FUNCTION_BLOCK ABSTRACT BaseCylinder IMPLEMENTS ITF_Cylinder
VAR_INPUT
END_VAR
VAR_OUTPUT
END_VAR
VAR
	//Hardware
	DI_Extended AT %I* : BOOL;
	DI_Retracted AT %I* : BOOL;
	DO_Extend AT %Q* : BOOL;
	//NOT USED BUT USABLE	
	DI_BoundaryPressure AT %I* : BOOL;
	DI_BoundaryFlowPressure AT %I* : BOOL;
	AI_PressureSensor AT %I* : INT;
	AI_FlowPressure AT %I* : INT;
	AI_PositionTransmitter AT %I* : INT;
END_VAR

PROPERTY Extended : BOOL
GET
Extended := DI_Extended;
END_GET
END_PROPERTY

METHOD ABSTRACT METH_Extend : BOOL
END_METHOD

METHOD ABSTRACT METH_Retract : BOOL
END_METHOD

PROPERTY Retracted : BOOL
GET
Retracted := DI_Retracted;
END_GET
END_PROPERTY

END_FUNCTION_BLOCK

(* stored: Version 1.1.0.1, ProductVersion 3.1.4024.9
   POU BaseCylinder: Id {0fc64f5a-1ee9-413f-9cbc-5836d5f79a93}, SpecialFunc None
   Property Extended: Id {283f46f2-b4ba-4a4c-89b0-c22d3a6bae68}
   Get Get: Id {b6f9aef2-3541-415c-90b5-e54255501b41}
   Method METH_Extend: Id {a919f99e-6a78-47eb-839b-1a0df0b366d7}
   Method METH_Retract: Id {23e0d501-f25e-416e-b5ed-b063d603a3a7}
   Property Retracted: Id {5700e9a8-67a6-40d5-ba2e-6a34df2ffd2a}
   Get Get: Id {b37b52dd-1411-4925-97db-c533348bcabc} *)
